Yaskawa INFORM job: SQUARE5.JBI

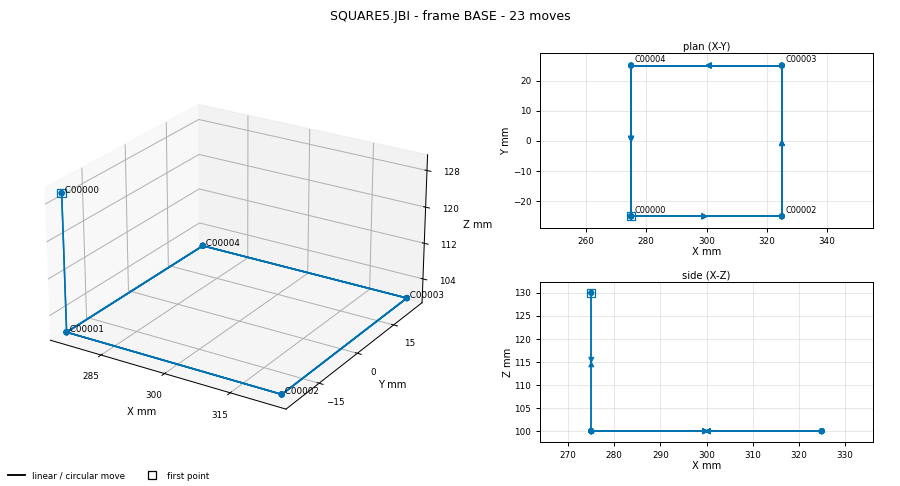
[picture p0: tool path of SQUARE5.JBI in frame BASE, 23 of 23 moves have a stored position in this frame; points joined in program order, loops and branches not executed]
/JOB
//NAME SQUARE5
//POS
///NPOS 6,0,0,0,0,0
///TOOL 0
///POSTYPE BASE
///RECTAN
C00000=275.000,-25.000,130.000,180.0000,0.0000,0.0000
C00001=275.000,-25.000,100.000,180.0000,0.0000,0.0000
C00002=325.000,-25.000,100.000,180.0000,0.0000,0.0000
C00003=325.000,25.000,100.000,180.0000,0.0000,0.0000
C00004=275.000,25.000,100.000,180.0000,0.0000,0.0000
C00005=275.000,-25.000,130.000,180.0000,0.0000,0.0000
//INST
///DATE 2026/04/01 12:00
///ATTR SC,RW
///GROUP1 RB1
NOP
SETTOOL TL#0
MOVJ C00000 VJ=5.00
MOVL C00001 V=100.0
MOVL C00002 V=100.0
MOVL C00003 V=100.0
MOVL C00004 V=100.0
MOVL C00001 V=100.0
MOVL C00002 V=100.0
MOVL C00003 V=100.0
MOVL C00004 V=100.0
MOVL C00001 V=100.0
MOVL C00002 V=100.0
MOVL C00003 V=100.0
MOVL C00004 V=100.0
MOVL C00001 V=100.0
MOVL C00002 V=100.0
MOVL C00003 V=100.0
MOVL C00004 V=100.0
MOVL C00001 V=100.0
MOVL C00002 V=100.0
MOVL C00003 V=100.0
MOVL C00004 V=100.0
MOVL C00001 V=100.0
MOVL C00005 V=100.0
END
